INTERFACE I_Component EXTENDS I_Base

METHOD Accept
VAR_INPUT
	ComponentVisitor : I_ComponentVisitor;
END_VAR
END_METHOD

METHOD DeregisterWithParent
VAR_INPUT
	Parent : I_ContainComponents;
END_VAR
END_METHOD

{attribute 'monitoring' := 'call'}
PROPERTY Name : T_MaxString
GET
END_GET
SET
END_SET
END_PROPERTY

METHOD RegisterWithParent
VAR_INPUT
	Parent : I_ContainComponents;
END_VAR
END_METHOD

END_INTERFACE

(* stored: Version 1.1.0.1, ProductVersion 3.1.4026.18
   Itf I_Component: Id {10547978-b502-4eff-be4f-753213a82870}
   Method Accept: Id {36a8d3c7-7340-416d-a0b4-669afb30e1f4}
   Method DeregisterWithParent: Id {7e9cd826-4c6e-4ffd-827b-e2e856690f75}
   Property Name: Id {cdc8512f-f17f-43fa-a89f-1cf233d832b2}
   Get Get: Id {8b62bfe2-6f79-4e0d-8061-9f86ed612e0f}
   Set Set: Id {e3081b5d-2401-42af-9fa8-188d7aa8aa07}
   Method RegisterWithParent: Id {3793a07f-c8e9-4833-b9d3-db0bbf855509} *)
